FUNCTION_BLOCK T_ExampleModule EXTENDS FB_PackML_BaseModule IMPLEMENTS I_ExampleEquipment

VAR
  
  cartesianRobot : T_ExampleEquipment;

  myProdMode : T_ExampleMOduleProductionMode;
  maintMode : T_ExampleMOduleProductionMode;
  manualMode : T_ExampleMOduleProductionMode;
 
  xAxis : yAxis, zAxis : T_Axis;
  grabber : T_Grabber;
  paramStruct : ST_ExampleParmas;
END_VAR

ComponentsCollection.AddComponent(xAxis);
ComponentsCollection.AddComponent(yAxis);
ComponentsCollection.AddComponent(zAxis);

SubModulesCollection.AddModule(grabber);
cartesianRobot.AddBits(
  xAxis := xAxis.GetRawAxis(),
  yAxis := yAxis,
  zAxis := zAxis,
  grabber := grabber);
  

paramsStruct.xAxis := xAxis;
paramStruct.yAxis := yAxis;
paramStruct.zAxis := zAxis;
paramStruct.grabber := grabber;


myProdMode.init(THIS^);

ModeManager.AddPackModes(myProdMode,maintMode,manualMode);
ModeManager.ChangeMode(E_PMLUnitMode.ePMLUnitMode_Production);

METHOD PUBLIC PickFromStagingArea : BOOL
VAR_INPUT
  orientationOfPick : ST_Orientation;
END_VAR
END_METHOD

END_FUNCTION_BLOCK

(* stored: Version 1.1.0.1, ProductVersion 3.1.4024.12
   POU T_ExampleModule: Id {b130e223-490b-4e61-95cf-3adea27f0c02}, SpecialFunc None
   Method PickFromStagingArea: Id {6209f71c-553e-4875-a5ac-3337e1fa137e} *)
